// TwinCAT 3 PLC project PnpComplexSolution
// ProgramVersion: 3.1.4024.12
// libraries:
//   Tc2_MC2, * (Beckhoff Automation GmbH)
//   Tc2_NcKinematicTransformation, * (Beckhoff Automation GmbH)
//   Tc2_Standard, * (Beckhoff Automation GmbH)
//   Tc2_System, * (Beckhoff Automation GmbH)
//   Tc3_Mc3Definitions, * (Beckhoff Automation GmbH)
//   Tc3_McCoordinatedMotion, * (Beckhoff Automation GmbH)
//   Tc3_Module, * (Beckhoff Automation GmbH)
// project tree:
//   DUTs/ StructFrame.TcDUT
//   GVLs/ GVL.TcGVL
//   / PlcTask.TcTTO (not stored)
//   POUs/ FB_AddAllAxes.TcPOU, FB_EnableAxes.TcPOU, FB_NCReset.TcPOU (not stored), MAIN.TcPOU
// real-time tasks:
//   TASK PlcTask: cycle T#10ms, priority 20, ADS port 350
//   TASK Job Task: cycle default, priority 32
// motion (NC):
//   TASK NC-Task 1 SAF: cycle T#2ms, priority 4, ADS port 501
//   TASK NC-Task 1 SVB: cycle T#10ms, priority 8, ADS port 511
//   AXIS ACS M1 (id 1)
//     Dynamic: Acceleration=1970.5, Deceleration=1970.5, Jerk=5911.5
//     Velo: RefSearch=13.1366666666667, RefSync=13.1366666666667, SlowManual=65.6833333333333, FastManual=394.1, Fast=1313.66666666667, Maximum=1313.66666666667
//     OtherSettings: AllowMotionCmdToSlave=true
//     encoder EncType=19
//       EncPara: ScaleFactorNumerator=70, ScaleFactorDenominator=1048576, Offset=6435.89, MaxCount=#xffffffff, ReferenceSystem=1
//         SoftEndMinControl: Range=320
//         SoftEndMaxControl: Range=460
//     drive DrvType=16
//       DrvPara: MaxCount=#xffffffff, DriveControlDWord=#x00020100
//         Analog: VeloReferenz=1445.03333333333, VeloScale=32, TorqueSetpointScale=10, ScaleFactorActTorque=0.1
//         TimeComp: TaskDelayCycles=1
//     controller CtrType=1
//       CtrPara: PriorControlFactor=1
//         Observer: BandWidth=20
//   AXIS ACS M2 (id 2)
//     Dynamic: Acceleration=2951.74, Deceleration=2951.74, Jerk=8855.22
//     Velo: RefSearch=19.6782762666667, RefSync=19.6782762666667, SlowManual=98.3913813333333, FastManual=590.348288, Fast=1967.82762666667, Maximum=1967.83
//     OtherSettings: AllowMotionCmdToSlave=true
//     encoder EncType=19
//       EncPara: ScaleFactorNumerator=104.8576, ScaleFactorDenominator=1048576, Offset=-203633.6, MaxCount=#xffffffff
//     drive DrvType=16
//       DrvPara: MaxCount=#xffffffff, DriveControlDWord=#x00020100
//         Analog: VeloReferenz=2164.61038933333, VeloScale=32, TorqueSetpointScale=10, ScaleFactorActTorque=0.1
//         TimeComp: TaskDelayCycles=1
//     controller CtrType=1
//       CtrPara: PriorControlFactor=1
//         Observer: BandWidth=20
//   AXIS ACS M3 (id 3)
//     Dynamic: Acceleration=2951.74, Deceleration=2951.74, Jerk=8855.22
//     Velo: RefSearch=19.6782762666667, RefSync=19.6782762666667, SlowManual=98.3913813333333, FastManual=590.348288, Fast=1967.82762666667, Maximum=1967.82762666667
//     OtherSettings: AllowMotionCmdToSlave=true
//     encoder EncType=19
//       EncPara: ScaleFactorNumerator=104.8576, ScaleFactorDenominator=1048576, Offset=-112438.85, MaxCount=#xffffffff
//     drive DrvType=16
//       DrvPara: MaxCount=#xffffffff, DriveControlDWord=#x00020100
//         Analog: VeloReferenz=2164.61038933333, VeloScale=32, TorqueSetpointScale=10, ScaleFactorActTorque=0.1
//         TimeComp: TaskDelayCycles=1
//     controller CtrType=1
//       CtrPara: PriorControlFactor=1
//         Observer: BandWidth=20
//   AXIS X (id 4)
//     Dynamic: Acceleration=2000, Deceleration=2000, Jerk=2000
//     OtherSettings: AllowMotionCmdToSlave=true
//     encoder EncType=1
//     drive DrvType=5
//       Analog: TorqueSetpointScale=10, ScaleFactorActTorque=0.1
//       TimeComp: TaskDelayCycles=1
//     controller CtrType=1
//       CtrPara: PriorControlFactor=1
//         Observer: BandWidth=20
//   AXIS Y (id 5)
//     Dynamic: Acceleration=2000, Deceleration=2000, Jerk=2000
//     OtherSettings: AllowMotionCmdToSlave=true
//     encoder EncType=1
//     drive DrvType=5
//       Analog: TorqueSetpointScale=10, ScaleFactorActTorque=0.1
//       TimeComp: TaskDelayCycles=1
//     controller CtrType=1
//       CtrPara: PriorControlFactor=1
//         Observer: BandWidth=20
//   AXIS Z (id 6)
//     Dynamic: Acceleration=2000, Deceleration=2000, Jerk=2000
//     OtherSettings: AllowMotionCmdToSlave=true
//     encoder EncType=1
//     drive DrvType=5
//       Analog: TorqueSetpointScale=10, ScaleFactorActTorque=0.1
//       TimeComp: TaskDelayCycles=1
//     controller CtrType=1
//       CtrPara: PriorControlFactor=1
//         Observer: BandWidth=20
// I/O:
//   DEVICE Device 2 (RT-Ethernet Adapter)
//   DEVICE Device 3 (EtherCAT), AmsNetId 5.37.99.176.4.1
//     Box 1 (CU2508) [CU2508 Ethernet Port]
//     Box 2 (EP7211-0034) [EP7211-0034 1Ch. MDP742 Servo motor output stage with OCT (50V, 4.5A RMS)]
//   DEVICE Device 4 (EtherCAT), AmsNetId 5.37.99.176.5.1
//     Box 3 (CU2508) [CU2508 Ethernet Port]
//     Box 4 (EP7211-0034) [EP7211-0034 1Ch. MDP742 Servo motor output stage with OCT (50V, 4.5A RMS)]
//   DEVICE Device 5 (EtherCAT), AmsNetId 5.37.99.176.6.1
//     Box 5 (CU2508) [CU2508 Ethernet Port]
//     Box 6 (EP7211-0034) [EP7211-0034 1Ch. MDP742 Servo motor output stage with OCT (50V, 4.5A RMS)]
//   DEVICE Device 1 (EtherCAT Automation Protocol), AmsNetId 5.37.99.176.2.1
//     Box 9 (Publisher)
//     Box 10 (Subscriber)
//   DEVICE Device 6 (EtherCAT), AmsNetId 5.37.99.176.7.1
//     Term 1 (EK1200) [EK1200-5000 EtherCAT Power supply (2A E-Bus)]
//       Term 8 (EL2004) [EL2004 4Ch. Dig. Output 24V, 0.5A]
//       Term 11 (EL9512) [EL9512 Power supply terminal 12V]
//       Term 12 (EL1904) [EL1904, 4 Ch. Safety Input 24V, TwinSAFE]
//         modules: Module 1 (FSOES)
//       Term 13 (EL2904) [EL2904, 4 Ch. Safety Output 24V, 0.5A, TwinSAFE]
//         modules: Module 1 (FSOES), Module 2 (DO)
//       Term 14 (EL1004) [EL1004 4Ch. Dig. Input 24V, 3ms]
//       Term 7 (EL9011) [EL9011 End Terminal]
// variable links:
//   NC-Task 1 SAF/Axes/ACS M1 <-> Device 3 (EtherCAT)/Box 2 (EP7211-0034)
//     Drive/Inputs/In/nDataIn1 <-> DRV Following error actual value/Following error actual value
//     Drive/Inputs/In/nDcOutputTime <-> InfoData/DcOutputShift
//     Drive/Inputs/In/nState1 <-> DRV Statusword/Statusword
//     Drive/Inputs/In/nState2 <-> DRV Statusword/Statusword @bit 8
//     Drive/Inputs/In/nState4 @bit 1 <-> WcState/InputToggle
//     Drive/Inputs/In/nState4 <-> WcState/WcState
//     Drive/Outputs/Out/nCtrl1 <-> DRV Controlword/Controlword
//     Drive/Outputs/Out/nCtrl2 <-> DRV Controlword/Controlword @bit 8
//     Drive/Outputs/Out/nDataOut1 <-> DRV Target position/Target position
//     Enc/Inputs/In/nDataIn1 <-> FB Position/Position
//     Enc/Inputs/In/nDcInputTime <-> InfoData/DcInputShift
//     Enc/Inputs/In/nState4 @bit 1 <-> WcState/InputToggle
//     Enc/Inputs/In/nState4 <-> WcState/WcState
//   NC-Task 1 SAF/Axes/ACS M2 <-> Device 4 (EtherCAT)/Box 4 (EP7211-0034)
//     Drive/Inputs/In/nDataIn1 <-> DRV Following error actual value/Following error actual value
//     Drive/Inputs/In/nDcOutputTime <-> InfoData/DcOutputShift
//     Drive/Inputs/In/nState1 <-> DRV Statusword/Statusword
//     Drive/Inputs/In/nState2 <-> DRV Statusword/Statusword @bit 8
//     Drive/Inputs/In/nState4 @bit 1 <-> WcState/InputToggle
//     Drive/Inputs/In/nState4 <-> WcState/WcState
//     Drive/Outputs/Out/nCtrl1 <-> DRV Controlword/Controlword
//     Drive/Outputs/Out/nCtrl2 <-> DRV Controlword/Controlword @bit 8
//     Drive/Outputs/Out/nDataOut1 <-> DRV Target position/Target position
//     Enc/Inputs/In/nDataIn1 <-> FB Position/Position
//     Enc/Inputs/In/nDcInputTime <-> InfoData/DcInputShift
//     Enc/Inputs/In/nState4 @bit 1 <-> WcState/InputToggle
//     Enc/Inputs/In/nState4 <-> WcState/WcState
//   NC-Task 1 SAF/Axes/ACS M3 <-> Device 5 (EtherCAT)/Box 6 (EP7211-0034)
//     Drive/Inputs/In/nDataIn1 <-> DRV Following error actual value/Following error actual value
//     Drive/Inputs/In/nDcOutputTime <-> InfoData/DcOutputShift
//     Drive/Inputs/In/nState1 <-> DRV Statusword/Statusword
//     Drive/Inputs/In/nState2 <-> DRV Statusword/Statusword @bit 8
//     Drive/Inputs/In/nState4 @bit 1 <-> WcState/InputToggle
//     Drive/Inputs/In/nState4 <-> WcState/WcState
//     Drive/Outputs/Out/nCtrl1 <-> DRV Controlword/Controlword
//     Drive/Outputs/Out/nCtrl2 <-> DRV Controlword/Controlword @bit 8
//     Drive/Outputs/Out/nDataOut1 <-> DRV Target position/Target position
//     Enc/Inputs/In/nDataIn1 <-> FB Position/Position
//     Enc/Inputs/In/nDcInputTime <-> InfoData/DcInputShift
//     Enc/Inputs/In/nState4 @bit 1 <-> WcState/InputToggle
//     Enc/Inputs/In/nState4 <-> WcState/WcState
//   PnpComplexSolution/PnpComplexSolution Instance <-> Device 1 (EtherCAT Automation Protocol)
//     PlcTask Inputs/MAIN.bEAP_DevState <-> Inputs/DevState
//   PnpComplexSolution/PnpComplexSolution Instance <-> Device 1 (EtherCAT Automation Protocol)/Box 10 (Subscriber)
//     PlcTask Inputs/MAIN.bEAP <-> bEAP/Inputs/VarData
//   PnpComplexSolution/PnpComplexSolution Instance <-> Device 1 (EtherCAT Automation Protocol)/Box 9 (Publisher)
//     PlcTask Outputs/MAIN.bReady <-> bReady/Outputs/VarData
//   PnpComplexSolution/PnpComplexSolution Instance <-> Device 6 (EtherCAT)/Term 1 (EK1200)/Term 8 (EL2004)
//     PlcTask Outputs/MAIN.bPlaceDone <-> Channel 1/Output
//   PnpComplexSolution/PnpComplexSolution Instance <-> NC-Task 1 SAF/Axes/ACS M1
//     PlcTask Inputs/GVL.stACSAxis[1].NcToPlc <-> Outputs/ToPlc
//     PlcTask Outputs/GVL.stACSAxis[1].PlcToNc <-> Inputs/FromPlc
//   PnpComplexSolution/PnpComplexSolution Instance <-> NC-Task 1 SAF/Axes/ACS M2
//     PlcTask Inputs/GVL.stACSAxis[2].NcToPlc <-> Outputs/ToPlc
//     PlcTask Outputs/GVL.stACSAxis[2].PlcToNc <-> Inputs/FromPlc
//   PnpComplexSolution/PnpComplexSolution Instance <-> NC-Task 1 SAF/Axes/ACS M3
//     PlcTask Inputs/GVL.stACSAxis[3].NcToPlc <-> Outputs/ToPlc
//     PlcTask Outputs/GVL.stACSAxis[3].PlcToNc <-> Inputs/FromPlc
//   PnpComplexSolution/PnpComplexSolution Instance <-> NC-Task 1 SAF/Axes/X
//     PlcTask Inputs/GVL.stAxis[1].NcToPlc <-> Outputs/ToPlc
//     PlcTask Outputs/GVL.stAxis[1].PlcToNc <-> Inputs/FromPlc
//   PnpComplexSolution/PnpComplexSolution Instance <-> NC-Task 1 SAF/Axes/Y
//     PlcTask Inputs/GVL.stAxis[2].NcToPlc <-> Outputs/ToPlc
//     PlcTask Outputs/GVL.stAxis[2].PlcToNc <-> Inputs/FromPlc
//   PnpComplexSolution/PnpComplexSolution Instance <-> NC-Task 1 SAF/Axes/Z
//     PlcTask Inputs/GVL.stAxis[3].NcToPlc <-> Outputs/ToPlc
//     PlcTask Outputs/GVL.stAxis[3].PlcToNc <-> Inputs/FromPlc
//   PnpComplexSolution/PnpComplexSolution Instance <-> NC-Task 1 SAF/Delta Robot
//     PlcTask Inputs/MAIN.in_stKinToPlc <-> Outputs/ToPlc
//     PlcTask Outputs/MAIN.out_stPlcToKin <-> Inputs/FromPlc
//   PnpComplexSolution/PnpComplexSolution Instance <-> NC-Task 1 SAF/Objects/Object1 (MC Group)
//     PlcTask Inputs/GVL.stGroupRef.NcToPlc <-> Group Outputs/ToPLC
//     PlcTask Outputs/GVL.stGroupRef.PlcToNc <-> Group Inputs/FromPLC

// ---- DUTs/StructFrame.TcDUT
TYPE StructFrame :
STRUCT
	rXpos : REAL := 0;
	rYpos : REAL := 0;
	rZpos : REAL := 0;
	sAlias : STRING := '';
END_STRUCT
END_TYPE

// ---- GVLs/GVL.TcGVL
VAR_GLOBAL
	stGroupRef			: AXES_GROUP_REF;
	stAxis				: ARRAY[1..cAxesCount] OF AXIS_REF;
	stACSAxis			: ARRAY[1..cAxesCount] OF AXIS_REF;
	PointAPos			: ARRAY[1..5,1..9] OF MC_LREAL;
	PointAPos2			: ARRAY[1..5,1..6] OF MC_LREAL;
	PointBPos			: ARRAY[1..5,1..9] OF MC_LREAL;
	MidPointPos			: ARRAY[1..3] OF MC_LREAL;
	PointAMidPos		: ARRAY[1..3] OF MC_LREAL;
	PointBMidPos		: ARRAY[1..3] OF MC_LREAL;
	PointXTSMidPos		: ARRAY[1..3] OF MC_LREAL;
	PreviousUpPos		: ARRAY[1..3] OF MC_LREAL;
	DeltaVelocity		: INT := 200;
	UpToMidBlend		: INT := 0;
	MidToUpBlend		: INT := 0;
	PointXTSPos			: ARRAY[1..6] OF MC_LREAL;
END_VAR

VAR_GLOBAL CONSTANT
	cAxesCount			: UINT:=3;
END_VAR

// ---- POUs/FB_AddAllAxes.TcPOU
FUNCTION_BLOCK FB_AddAllAxes
VAR_INPUT
	Execute				: BOOL;
END_VAR
VAR_OUTPUT
	Done				: BOOL;
	Busy				: BOOL;
	Error				: BOOL;
END_VAR
VAR
	fbAddAxis			: ARRAY[1..cAxesCount] OF MC_AddAxisToGroup;
	i					: UINT;
END_VAR

Done := TRUE;
Busy := FALSE;
Error := FALSE;

fbAddAxis[1].IdentInGroup := MCS_X; //X-Axis
fbAddAxis[2].IdentInGroup := MCS_Y; //Y-Axis
fbAddAxis[3].IdentInGroup := MCS_Z; //Z-Axis
fbAddAxis[4].IdentInGroup := MCS_C1;//1st rotation is C-rotation (around Z-Axis)

FOR i:=1 TO cAxesCount DO
	fbAddAxis[i](AxesGroup:=stGroupRef, Axis := stAxis[i], Execute := Execute);

	IF (NOT fbAddAxis[i].Done) THEN
		Done := FALSE;
	END_IF
	IF (fbAddAxis[i].Busy) THEN
		Busy := TRUE;
	END_IF
	IF (fbAddAxis[i].Error) THEN
		Error := TRUE;
	END_IF
END_FOR

END_FUNCTION_BLOCK

// ---- POUs/FB_EnableAxes.TcPOU
FUNCTION_BLOCK FB_EnableAxes
VAR_INPUT
	bEnableAxes: BOOL:= TRUE;
	fOverride:	LREAL	:= 100.0;
END_VAR
VAR_OUTPUT
	bAllAxesReady:	BOOL:= FALSE;
	Error: BOOL;
END_VAR
VAR_IN_OUT
	io_X:	AXIS_REF;
	io_Y:	AXIS_REF;
	io_Z:	AXIS_REF;
	io_C:	AXIS_REF;
	io_M1:	AXIS_REF;
	io_M2:	AXIS_REF;
	io_M3:	AXIS_REF;
END_VAR

VAR
	
	fbPowerX:	MC_Power;
	fbPowerY:	MC_Power;
	fbPowerZ:	MC_Power;
	fbPowerC:	MC_Power;
	fbPowerM1:	MC_Power;
	fbPowerM2:	MC_Power;
	fbPowerM3:	MC_Power;
END_VAR

io_X.ReadStatus();
io_Y.ReadStatus();
io_Z.ReadStatus();
io_C.ReadStatus();
io_M1.ReadStatus();
io_M2.ReadStatus();
io_M3.ReadStatus();


fbPowerX(
	Enable:=bEnableAxes, 
	Enable_Positive:=bEnableAxes, 
	Enable_Negative:=bEnableAxes, 
	Override:=fOverride, 
	BufferMode:= , 
	Axis:=io_X, 
	Status=> , 
	Busy=> , 
	Active=> , 
	Error=> , 
	ErrorID=> );
fbPowerY(
	Enable:=bEnableAxes, 
	Enable_Positive:=bEnableAxes, 
	Enable_Negative:=bEnableAxes, 
	Override:=fOverride, 
	BufferMode:= , 
	Axis:=io_Y, 
	Status=> , 
	Busy=> , 
	Active=> , 
	Error=> , 
	ErrorID=> );	
fbPowerZ(
	Enable:=bEnableAxes, 
	Enable_Positive:=bEnableAxes, 
	Enable_Negative:=bEnableAxes, 
	Override:=fOverride, 
	BufferMode:= , 
	Axis:=io_Z, 
	Status=> , 
	Busy=> , 
	Active=> , 
	Error=> , 
	ErrorID=> );	
fbPowerC(
	Enable:=bEnableAxes, 
	Enable_Positive:=bEnableAxes, 
	Enable_Negative:=bEnableAxes, 
	Override:=fOverride, 
	BufferMode:= , 
	Axis:=io_C, 
	Status=> , 
	Busy=> , 
	Active=> , 
	Error=> , 
	ErrorID=> );	
fbPowerM1(
	Enable:=bEnableAxes, 
	Enable_Positive:=bEnableAxes, 
	Enable_Negative:=bEnableAxes, 
	Override:=fOverride, 
	BufferMode:= , 
	Axis:=io_M1, 
	Status=> , 
	Busy=> , 
	Active=> , 
	Error=> , 
	ErrorID=> );	
fbPowerM2(
	Enable:=bEnableAxes, 
	Enable_Positive:=bEnableAxes, 
	Enable_Negative:=bEnableAxes, 
	Override:=fOverride, 
	BufferMode:= , 
	Axis:=io_M2, 
	Status=> , 
	Busy=> , 
	Active=> , 
	Error=> , 
	ErrorID=> );	
fbPowerM3(
	Enable:=bEnableAxes, 
	Enable_Positive:=bEnableAxes, 
	Enable_Negative:=bEnableAxes, 
	Override:=fOverride, 
	BufferMode:= , 
	Axis:=io_M3, 
	Status=> , 
	Busy=> , 
	Active=> , 
	Error=> , 
	ErrorID=> );	
bAllAxesReady	:= fbPowerX.Status AND fbPowerY.Status AND fbPowerZ.Status AND fbPowerC.Status AND 
	fbPowerM1.Status AND fbPowerM2.Status AND fbPowerM3.Status;
	
Error			:= fbPowerX.Error OR fbPowerY.Error OR fbPowerZ.Error OR fbPowerC.Error
	OR fbPowerM1.Error OR fbPowerM2.Error OR fbPowerM3.Error;

END_FUNCTION_BLOCK

// ---- POUs/MAIN.TcPOU
PROGRAM MAIN
VAR
	init : INT := 0;
END_VAR

HMILogic();
IF HMILogic.bRun = FALSE THEN
	Run.A_Man();
END_IF
IF HMILogic.bRun THEN
	Run(arrangedFrames := HMILogic.ArrangedFrames);
END_IF

END_PROGRAM
